// Mitsubishi GX Works2 project: z02   PLC: Q02/Q02H

PROGRAM MAIN
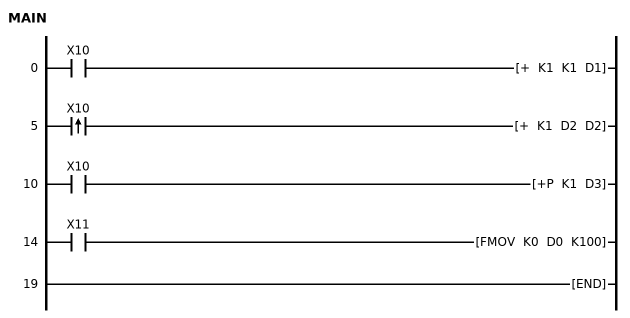
0     LD      X10
      +       K1 K1 D1
5     LDP     X10
      +       K1 D2 D2
10    LD      X10
      +P      K1 D3
14    LD      X11
      FMOV    K0 D0 K100
19    END
END_PROGRAM
